// LS Electric XG5000 project: Conveyer Controll with Sensor
// PLC LSPLC

PROGRAM NewProgram (task: 스캔 프로그램)

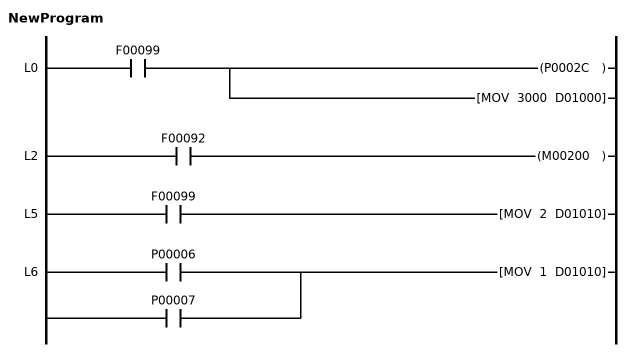
; L0
LOAD      F00099
OUT       P0002C
MOV       3000 D01000
; L2
LOAD      F00092
OUT       M00200
; L5
LOAD      F00099
MOV       2 D01010
; L6
LOAD      P00006
OR        P00007
MOV       1 D01010